Fanuc KAREL source: pos_clrpr.kl

PROGRAM pos_clrpr
%NOBUSYLAMP
%NOLOCKGROUP

VAR
	pr_num : INTEGER
%from tpe.klh %import get_int_arg
%from posetp.klh %import clrpr

BEGIN
	pr_num = tpe__get_int_arg(1)
	posetp__clrpr(pr_num)
END pos_clrpr
